// TIA Portal project "FactoryIO_Template_S7-1200_V15_V15.1" (V15.1)
// Vorlageprojekt für das Buch mit Zielsystem S7-1200

(* hardware
DEVICE "S7-1200-Station_1"  S7-1200 Station
   slot 0: "Baugruppenträger_0"  Rack  V1.0
   slot 1: "PLC_1"  CPU 1211C DC/DC/DC  6ES7 211-1AE40-0XB0  V4.1
DEVICE "HMI_1"  TP700 Comfort
   slot 0: "HMI_1"  TP700 Comfort  6AV2 124-0GC01-0AX0  15.1.0.0
   slot 1: "HMI_RT_1"  TP700 Comfort  6AV2 124-0GC01-0AX0  15.1.0.0
   slot 5: "HMI_1.IE_CP_1"  PROFINET Interface  15.0.1.0
      slot 1: "PROFINET Interface_1"  PROFINET Interface
         slot 1: "Port_1"  Port
         slot 2: "Port_2"  Port
   slot 7: "HMI_1.MPI/DP_CP_1"  MPI/DP Interface  15.0.1.0
*)

// ===== PLC "PLC_1"  CPU 1211C DC/DC/DC =====

VAR_GLOBAL   // PLC tag table "Standard-Variablentabelle"
   "Start" AT %I0.0 : Bool;
   "Stop" AT %I0.1 : Bool;
   "Reset" AT %I0.2 : Bool;
   "Estop" AT %I0.3 : Bool;
   "CB1" AT %I0.4 : Bool;
   "CB3" AT %I0.5 : Bool;
   "CB2" AT %I0.6 : Bool;
   "CB4" AT %I0.7 : Bool;
   "CB5" AT %I1.0 : Bool;
   "Auto" AT %I1.1 : Bool;
   "Manual" AT %I1.2 : Bool;
   "BT1" AT %Q0.0 : Bool;
   "BTM" AT %Q0.1 : Bool;
   "BTL" AT %Q0.2 : Bool;
   "BTS1" AT %Q0.3 : Bool;
   "BTS2" AT %Q0.4 : Bool;
   "BTVan" AT %Q0.5 : Bool;
   "BTXuat" AT %Q0.6 : Bool;
   "DStart" AT %Q0.7 : Bool;
   "DStop" AT %Q1.0 : Bool;
   "DReset" AT %Q1.1 : Bool;
   "DH" AT %Q1.2 : Bool;
   "DH Trai" AT %Q2.0 : Bool;
   "DH Phai" AT %Q2.1 : Bool;
   "BT CAN" AT %Q2.2 : Bool;
   "CB CAN" AT %ID32 : Real;
   "PTurn" AT %Q2.3 : Bool;
   "PPush" AT %Q2.4 : Bool;
   "PBelt" AT %Q2.5 : Bool;
   "PClam" AT %Q2.6 : Bool;
   "POpen" AT %Q2.7 : Bool;
   "Len" AT %Q3.0 : Bool;
   "Xuong" AT %Q3.1 : Bool;
   "ChayTheoHuong" AT %Q3.2 : Bool;
   "BTXich" AT %Q3.3 : Bool;
   "Mauto" AT %M0.0 : Bool;
   "MStart" AT %M0.2 : Bool;
   "MManual" AT %M0.1 : Bool;
   "MBT1" AT %M0.3 : Bool;
   "Tag_1" AT %M8.0 : Bool;
   "MRight" AT %M0.4 : Bool;
   "MLeft" AT %M0.5 : Bool;
   "MBT Can" AT %M0.6 : Bool;
   "KG" AT %MD9 : DInt;
   "CBXich(Truoc)" AT %I1.3 : Bool;
   "CBXich(Sau)" AT %I1.4 : Bool;
   "MCB5" AT %M0.7 : Bool;
   "CBPush" AT %I1.5 : Bool;
   "CBOpen" AT %I2.0 : Bool;
   "CBClam" AT %I2.1 : Bool;
   "Tag_2" AT %M8.1 : Bool;
   "Tag_3" AT %M8.2 : Bool;
   "MDonggoi" AT %M1.0 : Bool;
   "Tag_4" AT %M8.3 : Bool;
   "CBLenXuong" AT %I2.2 : Bool;
   "Tag_5" AT %M8.4 : Bool;
   "Tag_6" AT %M8.5 : Bool;
   "MResetOpen" AT %M1.2 : Bool;
   "MXich" AT %M1.3 : Bool;
   "Tag_7" AT %M8.6 : Bool;
   "Tag_8" AT %M1.4 : Bool;
   "Tag_9" AT %M2.0 : Bool;
   "Tag_10" AT %M3.0 : Bool;
   "Tag_11" AT %M3.1 : Bool;
   "Tag_12" AT %M3.2 : Bool;
   "M_DEN_START" AT %M7.0 : Bool;
   "M_DEN_STOP" AT %M7.1 : Bool;
   "M_DEN_RESET" AT %M7.2 : Bool;
   "Tag_13" AT %M7.3 : Bool;
   "Den_Bao" AT %Q1.3 : Bool;
   "Coi_Hu" AT %Q1.4 : Bool;
   "SPTRENPALLET" AT %QD32 : DInt;
   "CBDAT" AT %I1.6 : Bool;
   "SPDAT" AT %QD36 : DInt;
   "Tag_14" AT %M3.3 : Bool;
   "Tag_15" AT %M3.4 : Bool;
   "Tag_16" AT %M3.5 : Bool;
END_VAR

// folder: System blocks/Program resources

DATA_BLOCK "IEC_Counter_0_DB"   // DB1
{ S7_Optimized_Access := 'TRUE' }
AUTHOR : Simatic
FAMILY : IEC
NAME : CNTR
VERSION : 1.0
// stored: InstanceOfName IEC_COUNTER
"IEC_COUNTER"
BEGIN
END_DATA_BLOCK

DATA_BLOCK "IEC_Counter_0_DB_1"   // DB2
{ S7_Optimized_Access := 'TRUE' }
AUTHOR : Simatic
FAMILY : IEC
NAME : CNTR
VERSION : 1.0
// stored: InstanceOfName IEC_COUNTER
"IEC_COUNTER"
BEGIN
END_DATA_BLOCK

DATA_BLOCK "IEC_Timer_0_DB"   // DB3
{ S7_Optimized_Access := 'TRUE' }
AUTHOR : Simatic
FAMILY : IEC
NAME : IEC_TMR
VERSION : 1.0
// stored: InstanceOfName IEC_TIMER
"IEC_TIMER"
BEGIN
END_DATA_BLOCK

DATA_BLOCK "IEC_Timer_0_DB_1"   // DB4
{ S7_Optimized_Access := 'TRUE' }
AUTHOR : Simatic
FAMILY : IEC
NAME : IEC_TMR
VERSION : 1.0
// stored: InstanceOfName IEC_TIMER
"IEC_TIMER"
BEGIN
END_DATA_BLOCK

DATA_BLOCK "IEC_Timer_0_DB_2"   // DB5
{ S7_Optimized_Access := 'TRUE' }
AUTHOR : Simatic
FAMILY : IEC
NAME : IEC_TMR
VERSION : 1.0
// stored: InstanceOfName IEC_TIMER
"IEC_TIMER"
BEGIN
END_DATA_BLOCK

DATA_BLOCK "IEC_Timer_0_DB_3"   // DB6
{ S7_Optimized_Access := 'TRUE' }
AUTHOR : Simatic
FAMILY : IEC
NAME : IEC_TMR
VERSION : 1.0
// stored: InstanceOfName IEC_TIMER
"IEC_TIMER"
BEGIN
END_DATA_BLOCK

DATA_BLOCK "IEC_Timer_0_DB_4"   // DB7
{ S7_Optimized_Access := 'TRUE' }
AUTHOR : Simatic
FAMILY : IEC
NAME : IEC_TMR
VERSION : 1.0
// stored: InstanceOfName IEC_TIMER
"IEC_TIMER"
BEGIN
END_DATA_BLOCK

DATA_BLOCK "IEC_Timer_0_DB_5"   // DB8
{ S7_Optimized_Access := 'TRUE' }
AUTHOR : Simatic
FAMILY : IEC
NAME : IEC_TMR
VERSION : 1.0
// stored: InstanceOfName IEC_TIMER
"IEC_TIMER"
BEGIN
END_DATA_BLOCK

// folder: (top level)

FUNCTION "MHJ-PLC-Lab-Function-S71200" : Void   // FC9000, SCL
{ S7_Optimized_Access := 'TRUE' }
VERSION : 0.1
   VAR_TEMP
      rdTimeReturn : Int;
      outputTime : DTL;
      SyncVal : Byte;
      forVal : Int;
      forVal_2 : Int;
      Value : Byte;
   END_VAR
   VAR CONSTANT
      CompVal : Byte := 16#34;
      Value_01 : Byte := 16#11;
      Value_01_DW : DWord := 16#A165_D992;
      Value_02_DW : DWord := 16#58BE_4401;
   END_VAR
BEGIN

   #Value:=PEEK(area := 16#82,
        dbNumber := 0,
        byteOffset := 511);
   #Value := #Value + 1;

   POKE(area := 16#82,
        dbNumber := 0,
        byteOffset := 511,
        value := #Value);

   POKE(area:=16#81,
        dbNumber:=0,
        byteOffset:=1016,
        value:=#Value_01_DW);
   POKE(area := 16#81,
        dbNumber := 0,
        byteOffset := 1020,
        value := #Value_02_DW);

   POKE(area := 16#81,
        dbNumber := 0,
        byteOffset := 511,
        value := B#16#00);

   FOR #forVal := 0 TO 120 DO
       FOR #forVal_2:=0 TO 10 DO
           #rdTimeReturn:=RD_SYS_T(#outputTime);
           #rdTimeReturn := WR_SYS_T(#outputTime);
           #rdTimeReturn := RD_SYS_T(#outputTime);
           #rdTimeReturn := WR_SYS_T(#outputTime);
       END_FOR;
       #SyncVal:= PEEK(area := 16#81,
                      dbNumber := 0,
                      byteOffset := 511);
       IF #SyncVal = #CompVal THEN
          GOTO M_1;
       END_IF;
   END_FOR;
   RETURN;

   M_1:
   POKE(area := 16#81,
        dbNumber := 0,
        byteOffset := 511,
        value := B#16#0);
END_FUNCTION

ORGANIZATION_BLOCK "Main"   // OB1, LAD, ProgramCycle
TITLE = "Main Program Sweep (Cycle)"
{ S7_Optimized_Access := 'TRUE' }
VERSION : 0.1
   VAR_INPUT
      Initial_Call : Bool;   // Initial call of this OB
      Remanence : Bool;   // =True, if remanent data are available
   END_VAR
   VAR_TEMP   // added for the SCL form of the ladder/FBD networks
      _w1 : Bool;
      _w2 : Bool;
      _w3 : Bool;
   END_VAR
BEGIN

REGION Network 1: Konnektierungsbaustein für PLC-Lab
   // Im Netzwerk 1 wird der Konnektierungsbaustein für PLC-Lab aufgerufen.
   // Dieser Aufruf darf nicht entfernt werden!
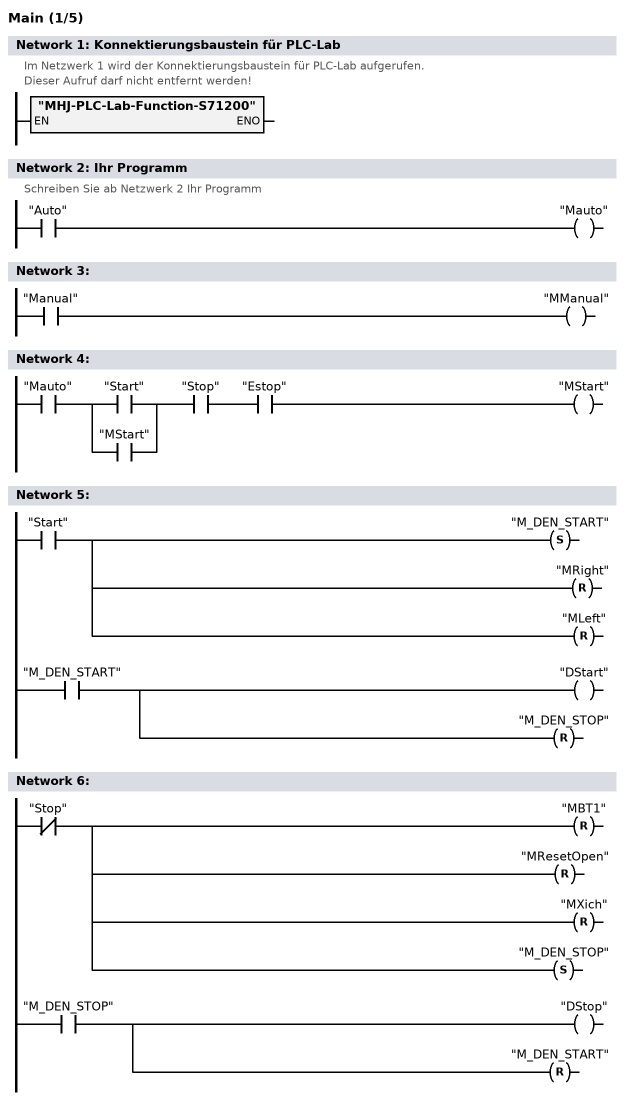
   RUNG wire#powerrail
      "MHJ-PLC-Lab-Function-S71200"()
   END_RUNG
   // the same network as SCL:
   "MHJ-PLC-Lab-Function-S71200"();
END_REGION

REGION Network 2: Ihr Programm
   // Schreiben Sie ab Netzwerk 2 Ihr Programm
   RUNG wire#powerrail
      Contact( "Auto" )
      Coil( "Mauto" )
   END_RUNG
   // the same network as SCL:
   "Mauto" := "Auto";
END_REGION

REGION Network 3
   RUNG wire#powerrail
      Contact( "Manual" )
      Coil( "MManual" )
   END_RUNG
   // the same network as SCL:
   "MManual" := "Manual";
END_REGION

REGION Network 4
   RUNG wire#powerrail
      Contact( "Mauto" )
      wire#w1
      Contact( "Start" )
      wire#w2
      Contact( "Stop" )
      Contact( "Estop" )
      Coil( "MStart" )
   END_RUNG
   RUNG wire#w1
      Contact( "MStart" )
   END_RUNG wire#w2
   // the same network as SCL:
   "MStart" := "Mauto" AND ("Start" OR "MStart") AND "Stop" AND "Estop";
END_REGION

REGION Network 5
   RUNG wire#powerrail
      Contact( "Start" )
      wire#w1
      S_Coil( "M_DEN_START" )
   END_RUNG
   RUNG wire#w1
      R_Coil( "MRight" )
   END_RUNG
   RUNG wire#w1
      R_Coil( "MLeft" )
   END_RUNG
   RUNG wire#powerrail
      Contact( "M_DEN_START" )
      wire#w2
      Coil( "DStart" )
   END_RUNG
   RUNG wire#w2
      R_Coil( "M_DEN_STOP" )
   END_RUNG
   // the same network as SCL:
   IF "Start" THEN
       "M_DEN_START" := TRUE;
       "MRight" := FALSE;
       "MLeft" := FALSE;
   END_IF;
   "DStart" := "M_DEN_START";
   IF "M_DEN_START" THEN "M_DEN_STOP" := FALSE; END_IF;
END_REGION

REGION Network 6
   RUNG wire#powerrail
      I_Contact( "Stop" )
      wire#w1
      R_Coil( "MBT1" )
   END_RUNG
   RUNG wire#w1
      R_Coil( "MResetOpen" )
   END_RUNG
   RUNG wire#w1
      R_Coil( "MXich" )
   END_RUNG
   RUNG wire#w1
      S_Coil( "M_DEN_STOP" )
   END_RUNG
   RUNG wire#powerrail
      Contact( "M_DEN_STOP" )
      wire#w2
      Coil( "DStop" )
   END_RUNG
   RUNG wire#w2
      R_Coil( "M_DEN_START" )
   END_RUNG
   // the same network as SCL:
   IF NOT "Stop" THEN
       "MBT1" := FALSE;
       "MResetOpen" := FALSE;
       "MXich" := FALSE;
       "M_DEN_STOP" := TRUE;
   END_IF;
   "DStop" := "M_DEN_STOP";
   IF "M_DEN_STOP" THEN "M_DEN_START" := FALSE; END_IF;
END_REGION

REGION Network 7
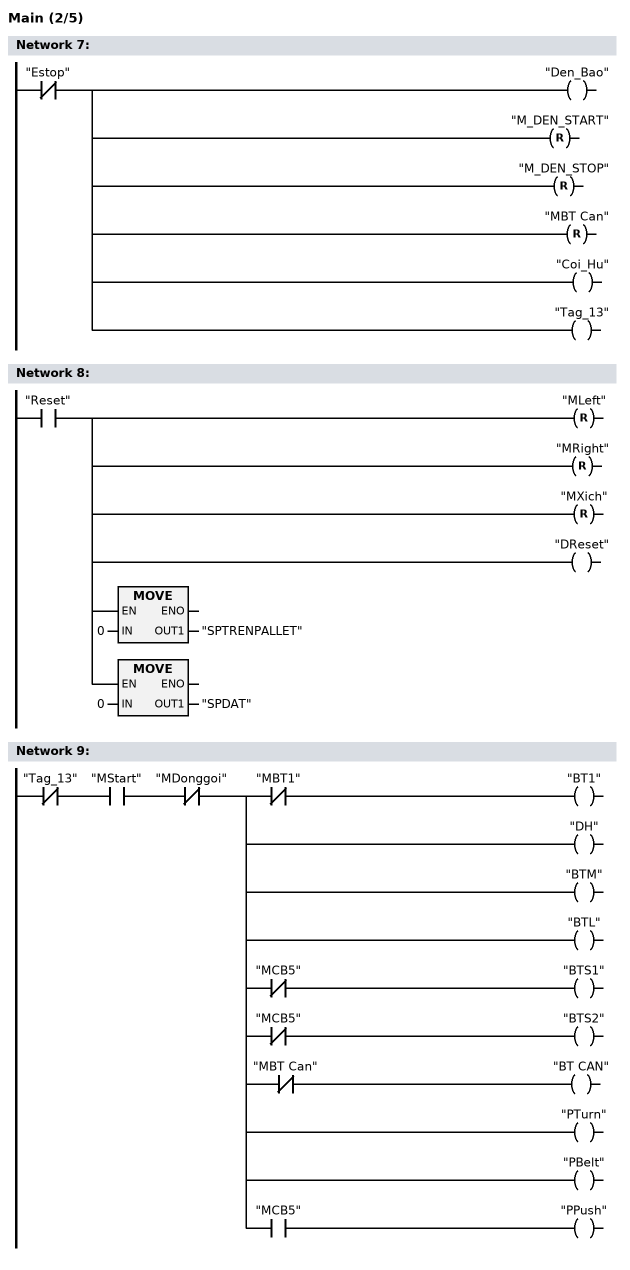
   RUNG wire#powerrail
      I_Contact( "Estop" )
      wire#w1
      Coil( "Den_Bao" )
   END_RUNG
   RUNG wire#w1
      R_Coil( "M_DEN_START" )
   END_RUNG
   RUNG wire#w1
      R_Coil( "M_DEN_STOP" )
   END_RUNG
   RUNG wire#w1
      R_Coil( "MBT Can" )
   END_RUNG
   RUNG wire#w1
      Coil( "Coi_Hu" )
   END_RUNG
   RUNG wire#w1
      Coil( "Tag_13" )
   END_RUNG
   // the same network as SCL:
   "Den_Bao" := NOT "Estop";
   IF NOT "Estop" THEN
       "M_DEN_START" := FALSE;
       "M_DEN_STOP" := FALSE;
       "MBT Can" := FALSE;
   END_IF;
   "Coi_Hu" := NOT "Estop";
   "Tag_13" := NOT "Estop";
END_REGION

REGION Network 8
   RUNG wire#powerrail
      Contact( "Reset" )
      wire#w1
      R_Coil( "MLeft" )
   END_RUNG
   RUNG wire#w1
      R_Coil( "MRight" )
   END_RUNG
   RUNG wire#w1
      R_Coil( "MXich" )
   END_RUNG
   RUNG wire#w1
      Coil( "DReset" )
   END_RUNG
   RUNG wire#w1
      Move(in := 0, out1 => "SPTRENPALLET")
   END_RUNG
   RUNG wire#w1
      Move(in := 0, out1 => "SPDAT")
   END_RUNG
   // the same network as SCL:
   IF "Reset" THEN
       "MLeft" := FALSE;
       "MRight" := FALSE;
       "MXich" := FALSE;
   END_IF;
   "DReset" := "Reset";
   IF "Reset" THEN
       "SPTRENPALLET" := 0;
       "SPDAT" := 0;
   END_IF;
END_REGION

REGION Network 9
   RUNG wire#powerrail
      I_Contact( "Tag_13" )
      Contact( "MStart" )
      I_Contact( "MDonggoi" )
      wire#w1
      I_Contact( "MBT1" )
      Coil( "BT1" )
   END_RUNG
   RUNG wire#w1
      Coil( "DH" )
   END_RUNG
   RUNG wire#w1
      Coil( "BTM" )
   END_RUNG
   RUNG wire#w1
      Coil( "BTL" )
   END_RUNG
   RUNG wire#w1
      I_Contact( "MCB5" )
      Coil( "BTS1" )
   END_RUNG
   RUNG wire#w1
      I_Contact( "MCB5" )
      Coil( "BTS2" )
   END_RUNG
   RUNG wire#w1
      I_Contact( "MBT Can" )
      Coil( "BT CAN" )
   END_RUNG
   RUNG wire#w1
      Coil( "PTurn" )
   END_RUNG
   RUNG wire#w1
      Coil( "PBelt" )
   END_RUNG
   RUNG wire#w1
      Contact( "MCB5" )
      Coil( "PPush" )
   END_RUNG
   // the same network as SCL:
   #_w1 := NOT "Tag_13" AND "MStart" AND NOT "MDonggoi";
   "BT1" := #_w1 AND NOT "MBT1";
   "DH" := #_w1;
   "BTM" := #_w1;
   "BTL" := #_w1;
   "BTS1" := #_w1 AND NOT "MCB5";
   "BTS2" := #_w1 AND NOT "MCB5";
   "BT CAN" := #_w1 AND NOT "MBT Can";
   "PTurn" := #_w1;
   "PBelt" := #_w1;
   "PPush" := #_w1 AND "MCB5";
END_REGION

REGION Network 10
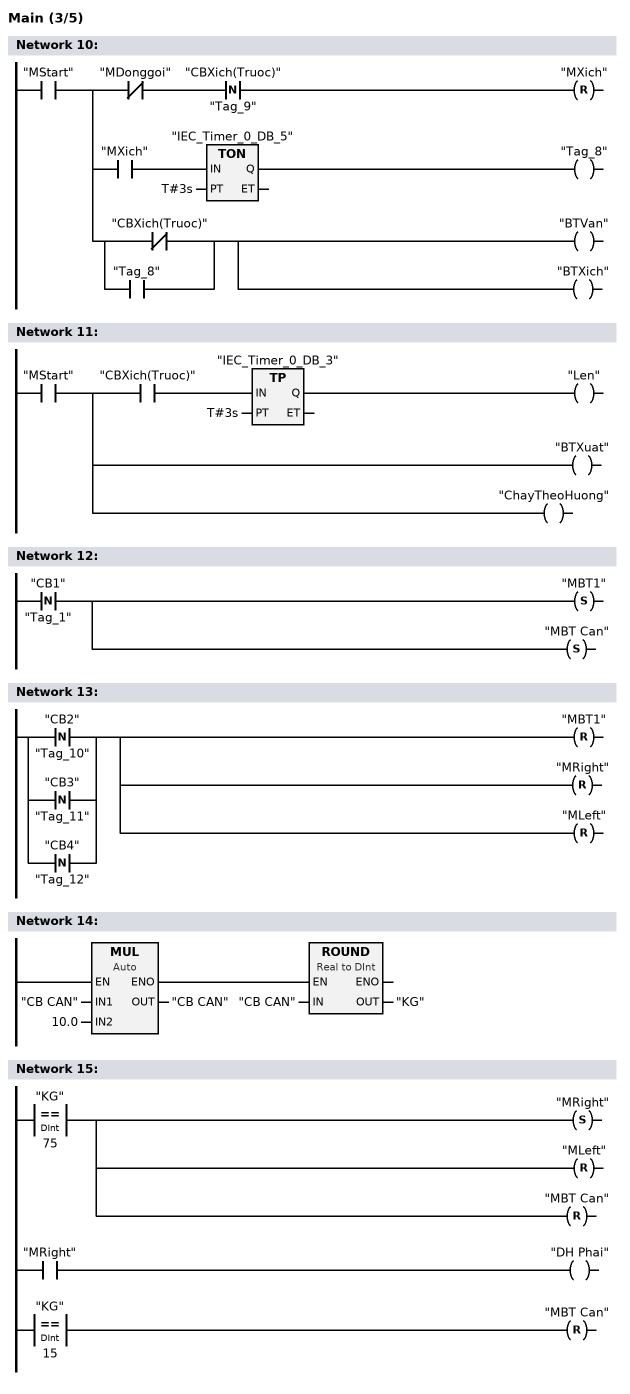
   #_w1 := "MStart" AND NOT "MDonggoi" AND NOT "CBXich(Truoc)" AND "Tag_9";   // falling edge of "CBXich(Truoc)"
   "Tag_9" := "CBXich(Truoc)";
   IF #_w1 THEN "MXich" := FALSE; END_IF;
   "IEC_Timer_0_DB_5".TON(IN := "MStart" AND "MXich", PT := T#3s);
   "Tag_8" := "IEC_Timer_0_DB_5".Q;
   "BTVan" := "MStart" AND (NOT "CBXich(Truoc)" OR "Tag_8");
   "BTXich" := "BTVan";
END_REGION

REGION Network 11
   "IEC_Timer_0_DB_3".TP(IN := "MStart" AND "CBXich(Truoc)", PT := T#3s);
   "Len" := "IEC_Timer_0_DB_3".Q;
   "BTXuat" := "MStart";
   "ChayTheoHuong" := "MStart";
END_REGION

REGION Network 12
   RUNG wire#powerrail
      N_Contact(operand := "CB1", bit := "Tag_1")
      wire#w1
      S_Coil( "MBT1" )
   END_RUNG
   RUNG wire#w1
      S_Coil( "MBT Can" )
   END_RUNG
   // the same network as SCL:
   #_w1 := NOT "CB1" AND "Tag_1";   // falling edge of "CB1"
   "Tag_1" := "CB1";
   IF #_w1 THEN
       "MBT1" := TRUE;
       "MBT Can" := TRUE;
   END_IF;
END_REGION

REGION Network 13
   RUNG wire#powerrail
      N_Contact(operand := "CB2", bit := "Tag_10")
      wire#w1
      R_Coil( "MBT1" )
   END_RUNG
   RUNG wire#powerrail
      N_Contact(operand := "CB3", bit := "Tag_11")
   END_RUNG wire#w1
   RUNG wire#powerrail
      N_Contact(operand := "CB4", bit := "Tag_12")
   END_RUNG wire#w1
   RUNG wire#w1
      R_Coil( "MRight" )
   END_RUNG
   RUNG wire#w1
      R_Coil( "MLeft" )
   END_RUNG
   // the same network as SCL:
   #_w1 := NOT "CB2" AND "Tag_10";   // falling edge of "CB2"
   "Tag_10" := "CB2";
   #_w2 := NOT "CB3" AND "Tag_11";   // falling edge of "CB3"
   "Tag_11" := "CB3";
   #_w3 := NOT "CB4" AND "Tag_12";   // falling edge of "CB4"
   "Tag_12" := "CB4";
   IF #_w1 OR #_w2 OR #_w3 THEN
       "MBT1" := FALSE;
       "MRight" := FALSE;
       "MLeft" := FALSE;
   END_IF;
END_REGION

REGION Network 14
   RUNG wire#powerrail
      Mul(in1 := "CB CAN", in2 := 10.0, out => "CB CAN")
      { S7_Templates := "[SrcType := Real, DestType := DInt]" } Round(in := "CB CAN", out => "KG")
   END_RUNG
   // the same network as SCL:
   "CB CAN" := "CB CAN" * 10.0;
   "KG" := ROUND("CB CAN");
END_REGION

REGION Network 15
   RUNG wire#powerrail
      { S7_Templates := "SrcType := DInt" } EQ_Contact(in1 := "KG", in2 := 75)
      wire#w1
      S_Coil( "MRight" )
   END_RUNG
   RUNG wire#w1
      R_Coil( "MLeft" )
   END_RUNG
   RUNG wire#w1
      R_Coil( "MBT Can" )
   END_RUNG
   RUNG wire#powerrail
      Contact( "MRight" )
      Coil( "DH Phai" )
   END_RUNG
   RUNG wire#powerrail
      { S7_Templates := "SrcType := DInt" } EQ_Contact(in1 := "KG", in2 := 15)
      R_Coil( "MBT Can" )
   END_RUNG
   // the same network as SCL:
   IF "KG" = 75 THEN
       "MRight" := TRUE;
       "MLeft" := FALSE;
       "MBT Can" := FALSE;
   END_IF;
   "DH Phai" := "MRight";
   IF "KG" = 15 THEN "MBT Can" := FALSE; END_IF;
END_REGION

REGION Network 16
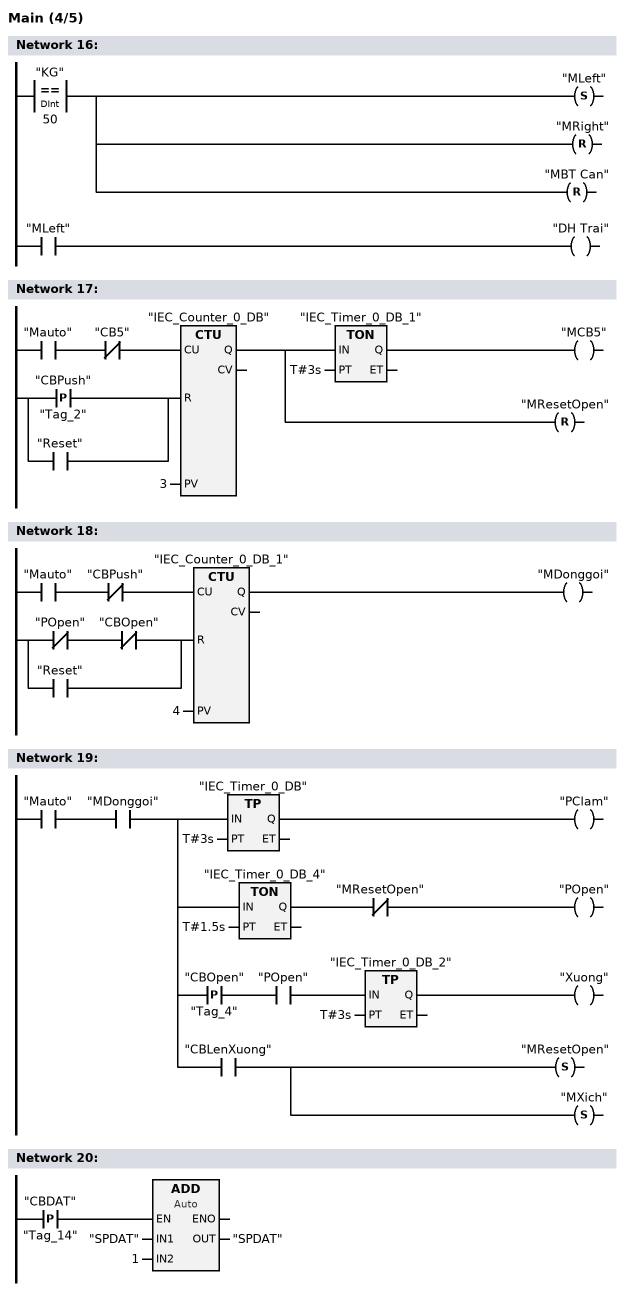
   RUNG wire#powerrail
      { S7_Templates := "SrcType := DInt" } EQ_Contact(in1 := "KG", in2 := 50)
      wire#w1
      S_Coil( "MLeft" )
   END_RUNG
   RUNG wire#w1
      R_Coil( "MRight" )
   END_RUNG
   RUNG wire#w1
      R_Coil( "MBT Can" )
   END_RUNG
   RUNG wire#powerrail
      Contact( "MLeft" )
      Coil( "DH Trai" )
   END_RUNG
   // the same network as SCL:
   IF "KG" = 50 THEN
       "MLeft" := TRUE;
       "MRight" := FALSE;
       "MBT Can" := FALSE;
   END_IF;
   "DH Trai" := "MLeft";
END_REGION

REGION Network 17
   #_w1 := "CBPush" AND NOT "Tag_2";   // rising edge of "CBPush"
   "Tag_2" := "CBPush";
   "IEC_Counter_0_DB".CTU(CU := "Mauto" AND NOT "CB5", R := #_w1 OR "Reset", PV := 3);
   "IEC_Timer_0_DB_1".TON(IN := "IEC_Counter_0_DB".Q, PT := T#3s);
   "MCB5" := "IEC_Timer_0_DB_1".Q;
   IF "IEC_Counter_0_DB".Q THEN "MResetOpen" := FALSE; END_IF;
END_REGION

REGION Network 18
   "IEC_Counter_0_DB_1".CTU(CU := "Mauto" AND NOT "CBPush",
                           R := (NOT "POpen" AND NOT "CBOpen") OR "Reset",
                           PV := 4);
   "MDonggoi" := "IEC_Counter_0_DB_1".Q;
END_REGION

REGION Network 19
   #_w1 := "Mauto" AND "MDonggoi";
   "IEC_Timer_0_DB".TP(IN := #_w1, PT := T#3s);
   "PClam" := "IEC_Timer_0_DB".Q;
   "IEC_Timer_0_DB_4".TON(IN := #_w1, PT := T#1.5s);
   "POpen" := "IEC_Timer_0_DB_4".Q AND NOT "MResetOpen";
   #_w2 := #_w1 AND "CBOpen" AND NOT "Tag_4";   // rising edge of "CBOpen"
   "Tag_4" := "CBOpen";
   "IEC_Timer_0_DB_2".TP(IN := #_w2 AND "POpen", PT := T#3s);
   "Xuong" := "IEC_Timer_0_DB_2".Q;
   IF #_w1 AND "CBLenXuong" THEN
       "MResetOpen" := TRUE;
       "MXich" := TRUE;
   END_IF;
END_REGION

REGION Network 20
   RUNG wire#powerrail
      P_Contact(operand := "CBDAT", bit := "Tag_14")
      Add(in1 := "SPDAT", in2 := 1, out => "SPDAT")
   END_RUNG
   // the same network as SCL:
   #_w1 := "CBDAT" AND NOT "Tag_14";   // rising edge of "CBDAT"
   "Tag_14" := "CBDAT";
   IF #_w1 THEN "SPDAT" := "SPDAT" + 1; END_IF;
END_REGION

REGION Network 21
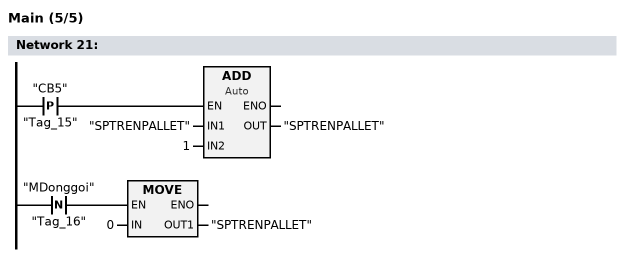
   RUNG wire#powerrail
      P_Contact(operand := "CB5", bit := "Tag_15")
      Add(in1 := "SPTRENPALLET", in2 := 1, out => "SPTRENPALLET")
   END_RUNG
   RUNG wire#powerrail
      N_Contact(operand := "MDonggoi", bit := "Tag_16")
      Move(in := 0, out1 => "SPTRENPALLET")
   END_RUNG
   // the same network as SCL:
   #_w1 := "CB5" AND NOT "Tag_15";   // rising edge of "CB5"
   "Tag_15" := "CB5";
   IF #_w1 THEN "SPTRENPALLET" := "SPTRENPALLET" + 1; END_IF;
   #_w2 := NOT "MDonggoi" AND "Tag_16";   // falling edge of "MDonggoi"
   "Tag_16" := "MDonggoi";
   IF #_w2 THEN "SPTRENPALLET" := 0; END_IF;
END_REGION
END_ORGANIZATION_BLOCK

(* ===== HMI "HMI_RT_1" =====
system functions are stored by id; their names below are inferred from use
connection "HMI_Connection_1": ETHERNET, S7_1200_OMS

HMI tags "Default tag table"
   "Tag_ScreenNumber" : UInt, internal

screen "Screen_1" 800x480
   TextField "Text field_1" at 208,17 size 400x110; Text 'BỘ GIÁO DỤC & ĐÀO TẠO TRƯỜNG ĐẠI HỌC SƯ PHẠM KỸ THUẬT TP. HỒ CHÍ MINH KHOA ĐIỆN – ĐIỆN TỬ BỘ MÔN TỰ ĐỘNG ĐIỀU KHIỂN'
   TextField "Text field_2" at 314,127 size 224x23; Text 'BÁO CÁO CUỐI KÌ'
   TextField "Text field_3" at 110,170 size 639x86; Text 'ĐỀ TÀI: ĐIỀU KHIỂN VÀ GIÁM SÁT MÔ HÌNH SẮP XẾP THEO KHỐI LƯỢNG BẰNG PLC'
   TextField "Text field_4" at 443,190 size 331x264; Text 'GVHD: TS. Trần Văn Sỹ Lớp PLCS330846_23_2_14 – Nhóm 1 SVTH MSSV Nguyễn Văn Pháp 21151303 Trần Minh Phúc 21151314 Võ Hưng Phát 21151308 Nguyễn Văn Qui 21151513 Nguyễn Hoài Thanh 21151335'
   Button "Button_1" at 7,437 size 134x31; TextOff 'ĐĂNG NHẬP'; TextOn 'Screen_2'
      on Click: ActivateScreen("Screen_2", 0)

screen "Screen_2" 800x480
   Button "Button_1" at 5,434 size 103x37; TextOff 'Home'; TextOn 'Screen_1'
      on Click: ActivateScreen("Screen_1", 0)
*)